(*********************************** G.D S.p.A. - Technical Department ***********************************
============= PROGRAM INFO ============
FOLDER:             TBD
MACHINES INVOLVED:  TBD 

============= DESCRIPTION =============
csp machine declaration

============= REVISIONS ===============
Date		Version	 	Author      	Description             
----------	-------		------------  	--------------------------------------------
2019/04/05 	0000.00	 	M.Grasso		Creation of the PRG

**********************************************************************************************************)
(*$R process_ref := prc; $*)
PROGRAM csp_case_flapControl_ls
VAR
	
	prc:											process;
	prc_path:										STRING;
	
END_VAR

_read_var_input();

_object_manager();

IF NOT objects_running()
THEN
	RETURN;	
END_IF

_read_process_image();

_mode_manager();

_set_runtime_properties();

(********************************* BODY *********************************)
(************************************************************************)

_handle_messages();

_write_output();

ACTION _handle_messages:
;
END_ACTION

ACTION _handle_process_test:
;
END_ACTION

ACTION _mode_manager:
IF process_mode_req_is_pending(prc)
THEN
    process_apply_mode_req_first_step(prc);
    CASE process_get_mode(prc) OF
        MODE_TO_ABSENT:
			;
        MODE_TO_INACTIVE:
			;
        MODE_TO_TEST:
			;
        MODE_TO_OPERATIONAL:
			;
    END_CASE
    process_apply_mode_req_second_step(prc);
END_IF
END_ACTION

ACTION _object_manager:
IF objects_initialization()
THEN
	sub_process_init(
		object_name					:= 'csp_case_flapControl_ls.prc', 
		process						:= csp_case_flapControl.prc, 
		CONVERSION_this				:= prc);
		
	prc_path 						:= process_get_path(prc);
END_IF

IF objects_running()
THEN
	process_cycle(prc);
END_IF
END_ACTION

ACTION _read_process_image:
;
END_ACTION

ACTION _read_var_input:
;
END_ACTION

ACTION _set_runtime_properties:
;
END_ACTION

ACTION _write_output:
;
END_ACTION

END_PROGRAM

(* stored: Version 1.1.0.1, ProductVersion 3.1.4022.12
   POU csp_case_flapControl_ls: Id {5d9a8ae1-51a2-44e1-ae30-353fc09e3cf7}, SpecialFunc None
   Action _handle_messages: Id {458b0286-a0b6-427f-b1f4-634adea62943}
   Action _handle_process_test: Id {5eba248b-553e-44ac-8b5a-f01c13a0bbf1}
   Action _mode_manager: Id {2a9bc9e5-bf16-414d-b41f-a4d55f443e93}
   Action _object_manager: Id {c52892ff-706d-4309-8522-123ce46fa44b}
   Action _read_process_image: Id {1afdba66-11a2-4158-a1ea-de0c2a1696ce}
   Action _read_var_input: Id {934be6fc-18da-4275-b0a0-ca0d1e79b628}
   Action _set_runtime_properties: Id {1d4ca6f1-fe1d-499a-95c2-fe34e44bc588}
   Action _write_output: Id {e4713f63-d998-4d84-89e2-29df38679f38} *)
